{attribute addProperty BoxType "EL3052-0000-0017"}
{attribute addProperty Id "AI_Standard_ChannelAT %I*ARRAY[0..1] OF AI_Standard_Channel_B51B79FC16220.250WcStateAT %I*WcState_F855686C1620InfoDataAT %I*InfoData_BC63D37F80100"}
{attribute addProperty CRC "3775335473"}
{attribute addProperty SizeInBites "258"}
{attribute addProperty SizeInBytes "32.25"}
TYPE EL3052_C3D795C5 :
STRUCT
	{attribute addProperty Name "AI_Standard_Channel"}
	AI_Standard_Channel : ARRAY[0..1] OF AI_Standard_Channel_B51B79FC;
	{attribute addProperty Name "WcState"}
	WcState : WcState_F855686C;
	{attribute addProperty Name "InfoData"}
	InfoData : InfoData_BC63D37F;
END_STRUCT
END_TYPE

(* stored: Version 1.2.0.0, ProductVersion 3.1.4024.9
   DUT EL3052_C3D795C5: Id {83edc4ab-7fc2-4146-af7b-0e8820494041} *)
